(* Logix 5000 project; controller Reto2 Emulate 5570 rev 30.12; software revision 30.00 *)

TASK MainTask (continuous, watchdog 500 ms) : MainProgram

MODULES
   Local : Emulate 5570 (ICP 2, rev 30.12)
END_MODULES

VAR_GLOBAL   (* controller tags *)
   BOX_AT_ENTRY : BOOL;   // Sensor cajas FactoryIO
   BOX_FEEDER : BOOL;   // Banda 1 cajas FactoryIO
   CLAMP : BOOL;   // Palanca junta cajas FactoryIO
   CLAMPED : BOOL;   // Sensor limite juntador FactoryIO
   CONTADOR_CAJAS : DINT;   // Display contador FactoryIO
   CONTADOR_PALLETS : DINT;
   CONTRAER_DE : BOOL;   // Piston Doble efecto Contraer Fisico
   ELEVATOR_DOWN : BOOL;   // Bajar elevador FactoryIO
   ELEVATOR_MOVING : BOOL;   // Sensor movimiento elevador FactoryIO
   ELEVATOR_UP : BOOL;   // Subir elevador FactoryIO
   EMERGENCY_STOP_FACTORY : BOOL;   // Boton stop emergency FactoryIO
   EXIT_CONVEYOR : BOOL;   // Banda 3 Pallet FactoryIO
   EXTENDER_DE : BOOL;   // Piston Doble efecto Extender Fisico
   EXTENDER_SE : BOOL;   // Piston Simple Efecto Fisico
   LOAD_BELT : BOOL;   // Banda 2 cajas FactoryIO
   LOAD_PALLET : BOOL;   // Banda 2 Pallet FactoryIO
   MOTORAC_FISICO : BOOL;   // Motor AC Fisico
   MOVE_TO_LIMIT : BOOL;   // Mover elevador al limite FactoryIO
   OPEN_PLATE : BOOL;   // Trampilla cajas FactoryIO
   PALLET_ENTRY : BOOL;   // Sensor 1 Pallet FactoryIO
   PALLET_EXIT : BOOL;   // Sensor 2 Pallet FactoryIO
   PALLET_FEEDER : BOOL;   // Banda 1 Pallet FactoryIO
   PALLET_LOADED : BOOL;
   PAUSED_FACTORYIO : BOOL;   // Pausando Sim FactoryIO
   PLATE_LIMIT : BOOL;   // Sensor limite compuerta FactoryIO
   PUSH : BOOL;   // Palanca empuja cajas Fisico
   PUSHER_LIMIT : BOOL;   // Sensor limite empujador FactoryIO
   RESET_FACTORYIO : BOOL;   // Boton reset FactoryIO
   RUNNING_FACTORYIO : BOOL;   // Ejecutando Sim FactoryIO
   START_FACTORYIO : BOOL;   // Boton verde FactoryIO
   START_FISICO : BOOL;   // Boton verde Fisico
   START_SCADA : BOOL;   // Boton verde SCADA
   STOP_FACTORYIO : BOOL;   // Boton rojo FactoryIO
   STOP_FISICO : BOOL;   // Boton rojo Fisico
   STOP_SCADA : BOOL;   // Boton rojo SCADA
   Temp : BOOL;
   TURN : BOOL;   // Palanca girar cajas FactoryIO
   WARNING_LIGHT : BOOL;   // Luces advertencia FactoryIO
END_VAR

PROGRAM MainProgram   (* main routine MainRoutine *)

ROUTINE MainRoutine   (* ladder *)
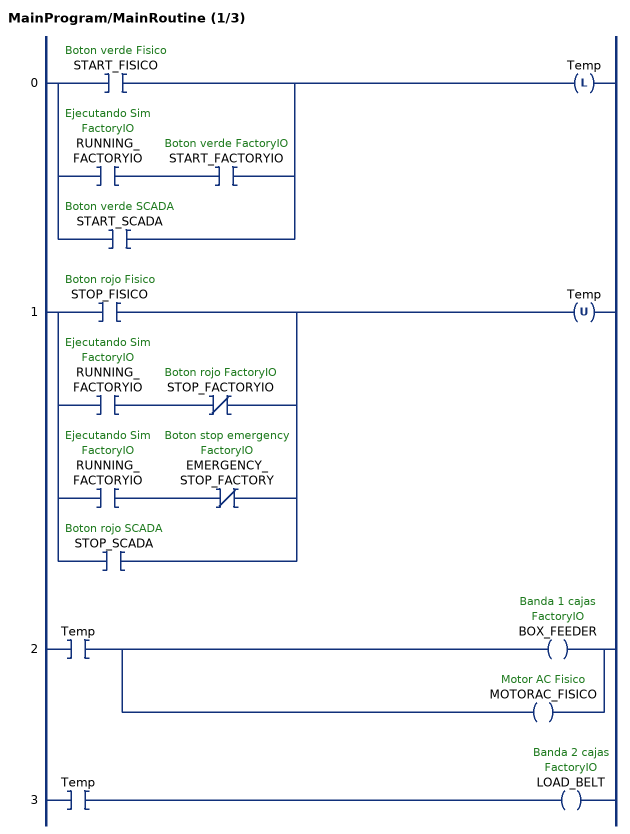
   0: [XIC(START_FISICO) ,[XIC(RUNNING_FACTORYIO) XIC(START_FACTORYIO) ,XIC(START_SCADA) ] ]OTL(Temp);
   1: [XIC(STOP_FISICO) ,[[XIC(RUNNING_FACTORYIO) XIO(STOP_FACTORYIO) ,XIC(RUNNING_FACTORYIO) XIO(EMERGENCY_STOP_FACTORY) ] ,XIC(STOP_SCADA) ] ]OTU(Temp);
   2: XIC(Temp)[OTE(BOX_FEEDER) ,OTE(MOTORAC_FISICO) ];
   3: XIC(Temp)OTE(LOAD_BELT);
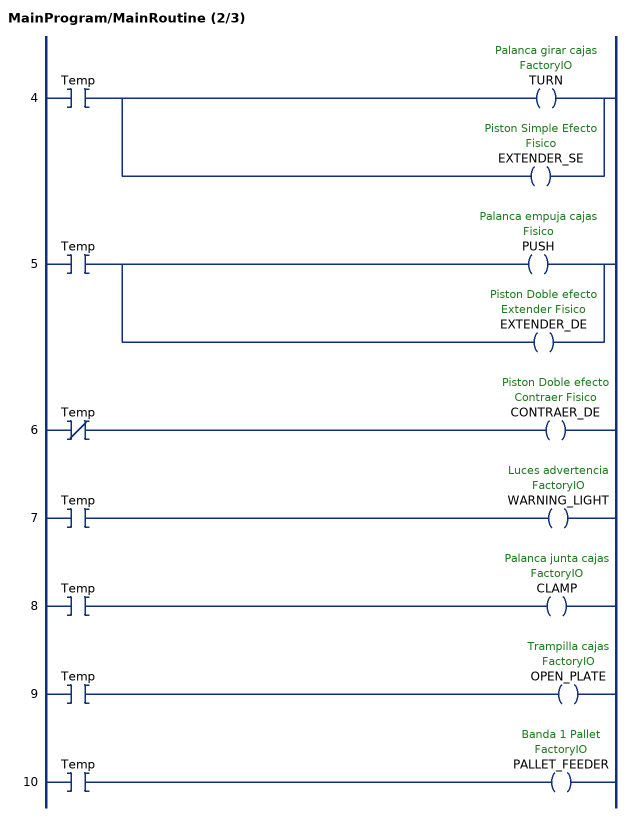
   4: XIC(Temp)[OTE(TURN) ,OTE(EXTENDER_SE) ];
   5: XIC(Temp)[OTE(PUSH) ,OTE(EXTENDER_DE) ];
   6: XIO(Temp)OTE(CONTRAER_DE);
   7: XIC(Temp)OTE(WARNING_LIGHT);
   8: XIC(Temp)OTE(CLAMP);
   9: XIC(Temp)OTE(OPEN_PLATE);
   10: XIC(Temp)OTE(PALLET_FEEDER);
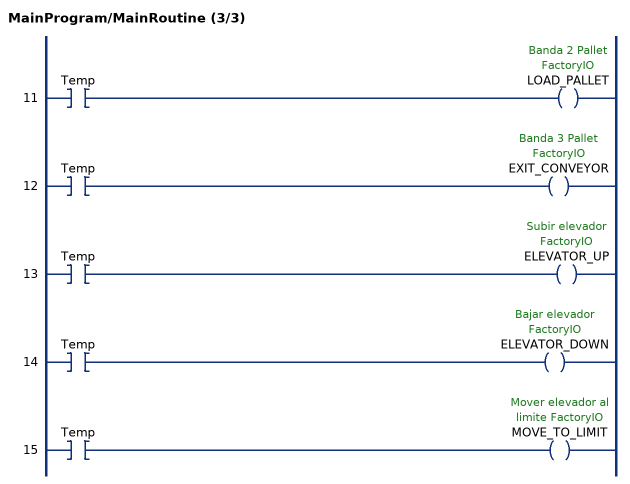
   11: XIC(Temp)OTE(LOAD_PALLET);
   12: XIC(Temp)OTE(EXIT_CONVEYOR);
   13: XIC(Temp)OTE(ELEVATOR_UP);
   14: XIC(Temp)OTE(ELEVATOR_DOWN);
   15: XIC(Temp)OTE(MOVE_TO_LIMIT);
END_ROUTINE
END_PROGRAM
